Fanuc KAREL source: IO0114.KL

-- PROVISIONAL review KL for V1013-1; original PC SHA256 2c9a3100f434a92948be1875d06c2ba98ed38b03afaf0443297d6428c7be3854
-- Incomplete behavior may be omitted. Consult companion uncertainty JSON. Do not deploy.
PROGRAM IO0114
%NOLOCKGROUP
-- UNRESOLVED_LOCAL_POOL 5 cells at code offset 13; source declarations unknown
-- DIRECT_LOCAL_WORD_ACCESS alone does not prove INTEGER, REAL, or BOOLEAN
BEGIN
  -- UNRESOLVED_PC offsets 0-18; opcodes 2B,2C,7B
  -- UNRESOLVED_PC offsets 23-30; opcodes 9D,23
  -- UNRESOLVED_PC offsets 35-49; opcodes 2E,22,9D,33,35
  -- UNRESOLVED_PC offsets 54-61; opcodes 9D,23
  -- UNRESOLVED_PC offsets 66-77; opcodes 2E,23
  -- UNRESOLVED_PC offsets 82-96; opcodes 21,19,23
  -- UNRESOLVED_PC offsets 101-105; opcodes 7F
  -- UNRESOLVED_PC offsets 110-114; opcodes 27,AA
  -- UNRESOLVED_PC offsets 119-123; opcodes 7F
END IO0114
